FUNCTION alg_M_example_controller_a_Dstopled : BOOL
VAR_INPUT
	state: STATE;
END_VAR

alg_M_example_controller_a_Dstopled := (((((((state.dvar_M_example_controller) <> (elit_wait_start)) AND ((state.dvar_M_example_controller) <> (elit_init2))) AND ((state.dvar_M_example_controller) <> (elit_droppoint))) AND ((state.dvar_M_example_controller) <> (elit_movetopickup))) AND ((state.dvar_M_example_controller) <> (elit_down))) AND ((state.dvar_M_example_controller) <> (elit_gopickup))) AND ((state.dvar_M_example_controller) <> (elit_goback));

END_FUNCTION

(* stored: Version 1.1.0.1, ProductVersion 3.1.4022.18
   POU alg_M_example_controller_a_Dstopled: Id {e33599b7-5eea-4e76-be6b-1f8c8af5c29b}, SpecialFunc None *)
